{attribute 'GeneratedUsingTerminal: EK1122-0000-0018'}
{attribute addProperty BoxType "EK1122-0000-0018"}
{attribute addProperty Id "Beckhoff_EKM1xxxsub_EK1100EK1100_1FC0878B2A_0001_EKM1101_0000_0016EKM1101_7F41762282A_0002_EKM1101_0000_0017EKM1101_7F41762282A_0003_EKM1101_0000_0018EKM1101_7F41762282A_0004_EKM1101_0000_0019EKM1101_7F41762282A_0005_EKM1101_0000_0020EKM1101_7F41762282"}
{attribute addProperty CRC "4030089381"}
{attribute addProperty Size "412"}
TYPE Beckhoff_EKM1xxxEK1122_F03648A5 EXTENDS EK1122_1FC0878B :
STRUCT
	{attribute addProperty Name "Beckhoff_EKM1xxxsub_EK1100"}
	{attribute addProperty PreviousPort "Beckhoff EKM1xxxEK1122 : D"}
	Beckhoff_EKM1xxxsub_EK1100 : EK1100_1FC0878B;
	{attribute addProperty Name "A_0001_EKM1101_0000_0016"}
	{attribute addProperty PreviousPort "Beckhoff EKM1xxxsub EK1100 : C"}
	A_0001_EKM1101_0000_0016 : EKM1101_7F417622;
	{attribute addProperty Name "A_0002_EKM1101_0000_0017"}
	{attribute addProperty PreviousPort "A_0001(EKM1101-0000-0016) : C"}
	A_0002_EKM1101_0000_0017 : EKM1101_7F417622;
	{attribute addProperty Name "A_0003_EKM1101_0000_0018"}
	{attribute addProperty PreviousPort "A_0002(EKM1101-0000-0017) : C"}
	A_0003_EKM1101_0000_0018 : EKM1101_7F417622;
	{attribute addProperty Name "A_0004_EKM1101_0000_0019"}
	{attribute addProperty PreviousPort "A_0003(EKM1101-0000-0018) : C"}
	A_0004_EKM1101_0000_0019 : EKM1101_7F417622;
	{attribute addProperty Name "A_0005_EKM1101_0000_0020"}
	{attribute addProperty PreviousPort "A_0004(EKM1101-0000-0019) : C"}
	A_0005_EKM1101_0000_0020 : EKM1101_7F417622;
END_STRUCT
END_TYPE

(* stored: Version 1.2.0.0, ProductVersion 3.1.4024.9
   DUT Beckhoff_EKM1xxxEK1122_F03648A5: Id {5c416b02-4586-42b6-a474-848f4edd5634} *)
